# EPICS autosave request: ipApp/Db/PACE5000_settings.req
$(P)$(R)Units
$(P)$(R)Setpoint
$(P)$(R)TweakVal
$(P)$(R)Slew
$(P)$(R)ReadSettingsScan.SCAN
